(* IEC 61131-3 sources: POMIRTS_lab3/AS/Library_2/AsHart, 3 files *)

(* ---- AsHart.typ ---- *)
TYPE
        hartIntState_t :
        (
           STATE_WAIT,
           STATE_WORK,
           STATE_FINISHED
        );
END_TYPE

(* ---- AsHart.fun ---- *)
{REDUND_CONTEXT} {REDUND_UNREPLICABLE} FUNCTION_BLOCK hartOpen (*open a device*)
	VAR_INPUT
		enable : BOOL; (*enables execution*)
		pDev : UDINT; (*device name given as a pointer to string*)
	END_VAR
	VAR_OUTPUT
		status : UINT; (*execution status: ERR_OK, ERR_FUB_ENABLE_FALSE, 0xXXXX = see help*)
		ident : UDINT; (*ident of the device*)
	END_VAR
	VAR
		_statemachine : hartIntState_t; (*internal variable*)
		_state : UINT; (*internal variable*)
	END_VAR
END_FUNCTION_BLOCK

{REDUND_CONTEXT} {REDUND_UNREPLICABLE} FUNCTION_BLOCK hartPutCmd (*put a command to a device*)
	VAR_INPUT
		enable : BOOL; (*enables execution*)
		ident : UDINT; (*ident of the device*)
		pCmd : UDINT; (*pointer to the command buffer*)
		cmdSize : UINT; (*size of command buffer*)
		pReply : UDINT; (*pointer to the reply buffer*)
		replySize : UINT; (*size of reply buffer*)
	END_VAR
	VAR_OUTPUT
		status : UINT; (*execution status: ERR_OK, ERR_FUB_ENABLE_FALSE, 0xXXXX = see help*)
		usedSize : UINT; (*used bytes in the read buffer*)
	END_VAR
	VAR
		_statemachine : hartIntState_t; (*internal variable*)
		_state : UINT; (*internal variable*)
		_pCmd : UDINT; (*internal variable*)
	END_VAR
END_FUNCTION_BLOCK

{REDUND_CONTEXT} {REDUND_UNREPLICABLE} FUNCTION_BLOCK hartClose (*close the device*)
	VAR_INPUT
		enable : BOOL; (*enables execution*)
		ident : UDINT; (*ident of the device*)
	END_VAR
	VAR_OUTPUT
		status : UINT; (*execution status: ERR_OK, ERR_FUB_ENABLE_FALSE, 0xXXXX = see help*)
	END_VAR
	VAR
		_statemachine : hartIntState_t; (*internal variable*)
		_state : UINT; (*internal variable*)
	END_VAR
END_FUNCTION_BLOCK

(* ---- AsHart.var ---- *)
(* error area 35580 - 35599 for AsHart reserved *)

VAR CONSTANT
	hartERR_INVALID_DEVICE		: UINT := 35580;
	hartERR_MODULE_DOESNT_EXIST	: UINT := 35581;
	hartERR_ALREADY_OPENED		: UINT := 35582;
	hartERR_DEVICE_OPEN		: UINT := 35583;
	hartERR_INVALID_IDENT		: UINT := 35584;
        hartERR_INVALID_BUFFER          : UINT := 35585;
	hartERR_PUT_CMD_IOCTL		: UINT := 35586;
	hartERR_QUEUE_FULL		: UINT := 35587;
	hartERR_DEVICE_CLOSE		: UINT := 35588;
END_VAR
